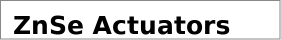
VISUALIZATION VISU_HMI_ZNSE_ACTUATORS  // 281x40
    Label (10,10 271x30), "ZnSe Actuators"
END_VISUALIZATION

(* stored: Version 1.1.0.1, ProductVersion 3.1.4024.14
   Visu VISU_HMI_ZNSE_ACTUATORS: Id {07542d35-27cb-4636-8341-d2e66bb2f067} *)
